KUKA KRL program: ini.src

&ACCESS RV1
&REL 14
&COMMENT INICIALIZACION E_S A PLC
&PARAM EDITMASK = *
&PARAM TEMPLATE = C:\KRC\Roboter\Template\vorgabe
DEF ini( )
;################################################
; PROYECTO: MAFELEC PLANTA DE BATERIAS
; ROBOT: 121_R1
; PROGRAMA: INICIALIZACION SENALES PLC
; CREADO POR: OBY-Wan Kenoby(zaisor robotics)
; FECHA: 23-NOVIEMBRE-2022
; MODIFICADO POR:
; FECHA MODIFICACION: 10-ENERO-2023
;################################################

Repite=0
$OUT[63]=FALSE  ; VOLVEMOS A CONTROLAR POR PLC EL SENSOR DE SOBREPASO
O_AREL_1=TRUE
O_AREL_2=TRUE
O_AREL_3=TRUE
O_AREL_4=TRUE
O_AREL_5=TRUE
O_AREL_6=TRUE
O_AREL_7=TRUE
O_AREL_8=TRUE


O_CREL_1=TRUE
O_CREL_2=TRUE
O_CREL_3=TRUE
O_CREL_4=TRUE
O_CREL_5=TRUE
O_CREL_6=TRUE
O_CREL_7=TRUE
O_CREL_8=TRUE


O_JRDY_1=FALSE
O_JRDY_2=FALSE
O_JRDY_3=FALSE
O_JRDY_4=FALSE
O_JRDY_5=FALSE
O_JRDY_6=FALSE
O_JRDY_7=FALSE
O_JRDY_8=FALSE

O_TREQ_1=FALSE
O_TREQ_2=FALSE
O_TREQ_3=FALSE
O_TREQ_4=FALSE
O_TREQ_5=FALSE
O_TREQ_6=FALSE
O_TREQ_7=FALSE
O_TREQ_8=FALSE

O_SERVPOS=FALSE
O_TYPE_RQ=FALSE

O_INPICKER_OK=FALSE
O_INPICKER_NOK=FALSE
O_ERR_VISION=FALSE

O_TYPE_INFO=0
FINALIZA=FALSE
FINALIZA_AZUL=FALSE
FINALIZA_VERDE=FALSE
SELECT_CELL=TRUE
SELECT_NEXT=FALSE
SELECT_T1=FALSE

INPICKER_Handler.DataToSend.command=0

O_LIMITS_OK=FALSE
O_LIMITS_NOK=FALSE

O_LIMIT_X=FALSE
O_LIMIT_Y=FALSE
O_LIMIT_Z=FALSE
O_LIMIT_A=FALSE
O_LIMIT_B=FALSE
O_LIMIT_C=FALSE

LIM_X=FALSE
LIM_Y=FALSE
LIM_Z=FALSE
LIM_A=FALSE
LIM_B=FALSE
LIM_C=FALSE

GIRO_A_P=FALSE
GIRO_A_N=FALSE
GIRO_B_P=FALSE
GIRO_B_N=FALSE
GIRO_C_P=FALSE
GIRO_C_N=FALSE

$TIMER[20]=0
$TIMER_STOP[20]=TRUE

$OUT[61]=FALSE

END
